# EPICS substitutions: evrSupport/Db/bsa/bsaProcTestAll.substitutions
file bsaProcTest.db
{
#             Meas Defn
#	            Name
  pattern { DEV      , MD,  MDID, LOCA       }
	      {  $(DEVICE)  , 1,   1, $(LOC)     }
	      {  $(DEVICE)  , 2,   2, $(LOC)     }
	      {  $(DEVICE)  , 3,   3, $(LOC)     }
	      {  $(DEVICE)  , 4,   4, $(LOC)     }
	      {  $(DEVICE)  , 5,   5, $(LOC)     }
	      {  $(DEVICE)  , 6,   6, $(LOC)     }
	      {  $(DEVICE)  , 7,   7, $(LOC)     }
	      {  $(DEVICE)  , 8,   8, $(LOC)     }
	      {  $(DEVICE)  , 9,   9, $(LOC)     }
	      {  $(DEVICE)  ,10,   10, $(LOC)    }
	      {  $(DEVICE)  ,11,   11, $(LOC)    }
	      {  $(DEVICE)  ,12,   1H, $(LOC)    }
	      {  $(DEVICE)  ,13,   TH, $(LOC)    }
	      {  $(DEVICE)  ,14,   BR, $(LOC)    }
	      {  $(DEVICE)  ,15,   CUS1H, $(LOC)    }
	      {  $(DEVICE)  ,16,   CUSTH, $(LOC)    }
	      {  $(DEVICE)  ,17,   CUSBR, $(LOC)    }
	      {  $(DEVICE)  ,18,   CUH1H, $(LOC)    }
	      {  $(DEVICE)  ,19,   CUHTH, $(LOC)    }
	      {  $(DEVICE)  ,20,   CUHBR, $(LOC)    }
}
